PROGRAM MAIN
VAR
	Counter	AT%Q*:UINT;
	fbSinWave	:FB_CTRL_SIGNAL_GENERATOR;
	Param: ST_CTRL_SIGNAL_GENERATOR_PARAMS := (tCtrlCycleTime := TIME#10ms, tTaskCycleTime := TIME#10ms, tCylceDuration := TIME#2s0ms, fAmplitude := 1000);
END_VAR

fbSinWave( 
	eMode:=E_CTRL_MODE.eCTRL_MODE_ACTIVE , 
	stParams:=Param );
	
	
Counter:=TO_UINT(fbSinWave.fOut);

END_PROGRAM

(* stored: Version 1.1.0.1, ProductVersion 3.1.4026.18
   POU MAIN: Id {cba2def1-e2df-437a-aa4b-e380efd05e6e}, SpecialFunc None *)
